// TIA Portal V21 export
TYPE "LBC_typeAxisControlNodeCommands"
TITLE = LBC_typeAxisControlNodeCommands
// Control Node Wapper commands
   STRUCT
      enableAxis { ExternalAccessible := 'False'; ExternalVisible := 'False'; ExternalWritable := 'False'} : Bool;   // Set axis enable
      resetAxis { ExternalAccessible := 'False'; ExternalVisible := 'False'; ExternalWritable := 'False'} : Bool;   // Rising edge: Acknowledgement of technology alarms or restart of the axis (depending on configuration)
      openBrake { ExternalAccessible := 'False'; ExternalVisible := 'False'; ExternalWritable := 'False'} : Bool;   // Unconditionally open brake
      jogForward { ExternalAccessible := 'False'; ExternalVisible := 'False'; ExternalWritable := 'False'} : Bool;   // Rising edge: Move an axis in jog mode (forward); Falling edge: Stop jogging
      jogBackward { ExternalAccessible := 'False'; ExternalVisible := 'False'; ExternalWritable := 'False'} : Bool;   // Rising edge: Move an axis in jog mode (backward); Falling edge: Stop jogging
      moveVelocity { ExternalAccessible := 'False'; ExternalVisible := 'False'; ExternalWritable := 'False'} : Bool;   // Rising edge: Move an axis at constant velocity/speed
      stop { ExternalAccessible := 'False'; ExternalVisible := 'False'; ExternalWritable := 'False'} : Bool;   // Rising edge: Brake an axis until it comes to a standstill. Note: MC_Halt is triggered internally
      fastStop { ExternalAccessible := 'False'; ExternalVisible := 'False'; ExternalWritable := 'False'} : Bool;   // Rising edge: Brake an axis until it comes to a standstill (with fastStop dynamics). Note: MC_Halt is triggered internally
      torqueLimiting { ExternalAccessible := 'False'; ExternalVisible := 'False'; ExternalWritable := 'False'} : Bool;   // Enable force/torque limiting
      homing { ExternalAccessible := 'False'; ExternalVisible := 'False'; ExternalWritable := 'False'} : Bool;   // Rising edge: Home axis
      posRelative { ExternalAccessible := 'False'; ExternalVisible := 'False'; ExternalWritable := 'False'} : Bool;   // Rising edge: Move an axis relative to its position when execution of the job began
      posAbsolute { ExternalAccessible := 'False'; ExternalVisible := 'False'; ExternalWritable := 'False'} : Bool;   // Rising edge: Move an axis to an absolute position
      posSuperimposed { ExternalAccessible := 'False'; ExternalVisible := 'False'; ExternalWritable := 'False'} : Bool;   // Rising edge: Start a superimposed positioning
      haltSuperimposed { ExternalAccessible := 'False'; ExternalVisible := 'False'; ExternalWritable := 'False'} : Bool;   // Manual superimposed halting from HMI, Rising edge: Decelerate a superimposed motion to zero velocity
      gearInRelative { ExternalAccessible := 'False'; ExternalVisible := 'False'; ExternalWritable := 'False'} : Bool;   // Rising edge: Start a gearing operation (relative)
      gearInAbsolute { ExternalAccessible := 'False'; ExternalVisible := 'False'; ExternalWritable := 'False'} : Bool;   // Rising edge: Start a gearing operation (absolute)
      gearInVelocity { ExternalAccessible := 'False'; ExternalVisible := 'False'; ExternalWritable := 'False'} : Bool;   // Manual velocity synchronous gearing from HMI, Rising edge: Start a gearing operation (velocity synchronous)
      camIn { ExternalAccessible := 'False'; ExternalVisible := 'False'; ExternalWritable := 'False'} : Bool;   // Rising edge: Start a camming operation
      gearOutCamOut { ExternalAccessible := 'False'; ExternalVisible := 'False'; ExternalWritable := 'False'} : Bool;   // Manual gearing/camming out operation from HMI, Rising edge: End gearing / camming operation
      phasing { ExternalAccessible := 'False'; ExternalVisible := 'False'; ExternalWritable := 'False'} : Bool;   // Rising edge: Start a phasing operation
      offset { ExternalAccessible := 'False'; ExternalVisible := 'False'; ExternalWritable := 'False'} : Bool;   // Manual offset operation from HMI, Rising edge: Start an offset operation (shift following value of an existing synchronous operation)
      reset { ExternalAccessible := 'False'; ExternalVisible := 'False'; ExternalWritable := 'False'} : Bool;   // Reinitialiazing the block
   END_STRUCT;
END_TYPE
